Staubli VAL3: template.pjx

Parameters version=s7.2.1 stackSize=5000 millimeterUnit=true
Data file=template.dtx
